// TIA Portal V20 export
TYPE "type_emRelations_em3_cmStatus"
// stored: Access Published, Namespace Unit1
   STRUCT
      cmSafetyPinIdlePositionSensor { S7_SetPoint := 'True'} : "LBC_typeDigitalSignalControlNode";
      cmRotationSafetyPinPositionSensor { S7_SetPoint := 'True'} : "LBC_typeDigitalSignalControlNode";
      cmIonizerTopMaintDetection { ExternalAccessible := 'False'; ExternalVisible := 'False'; ExternalWritable := 'False'} : "LBC_typeDigitalSignalControlNode";
      cmIonizerTopErrorDetection { ExternalWritable := 'False'} : "LBC_typeDigitalSignalControlNode";
      cmIonizerBtmMaintDetection { ExternalAccessible := 'False'; ExternalVisible := 'False'; ExternalWritable := 'False'; S7_SetPoint := 'True'} : "LBC_typeDigitalSignalControlNode";
      cmIonizerBtmErrorDetection { ExternalAccessible := 'False'; ExternalVisible := 'False'; ExternalWritable := 'False'; S7_SetPoint := 'True'} : "LBC_typeDigitalSignalControlNode";
      cmDancerEncoder { ExternalAccessible := 'False'; ExternalVisible := 'False'; ExternalWritable := 'False'} : "LBC_typeAnalogInputControlNode";
      cmLoadCellControllerInterface { S7_SetPoint := 'True'} : "LBC_typeAnalogInputControlNode";
      cmDancerElectroPneumaticRegulator { S7_SetPoint := 'True'} : "LBC_typeAnalogOutputControlNode";
      cmCompensatorAxisX { S7_SetPoint := 'True'} : "LBC_typeAxis64PosControlNode";
      cmMasterVirtualAxis { S7_SetPoint := 'True'} : "LBC_typeAxis64PosControlNode";
      cmUnwinderVirtualAxis { S7_SetPoint := 'True'} : "LBC_typeAxis64PosControlNode";
      cmDancerFwdBwd { S7_SetPoint := 'True'} : "LBC_typeTwoWayActuatorControlNode";
      cmSepaUnwinderIonizerTop { S7_SetPoint := 'True'} : "LBC_typeTwoWayActuatorControlNode";
      cmSepaUnwinderIonizerBottom { S7_SetPoint := 'True'} : "LBC_typeTwoWayActuatorControlNode";
      cmEpcPivot { S7_SetPoint := 'True'} : "LER_typeCON600ControlNode";
   END_STRUCT;
   // cmSafetyPinIdlePositionSensor.commands.reset := FALSE;
   // cmSafetyPinIdlePositionSensor.commands.simulation := FALSE;
   // cmSafetyPinIdlePositionSensor.commands.quality := TRUE;
   // cmRotationSafetyPinPositionSensor.commands.reset := FALSE;
   // cmRotationSafetyPinPositionSensor.commands.simulation := FALSE;
   // cmRotationSafetyPinPositionSensor.commands.quality := TRUE;
END_TYPE
